{attribute 'GeneratedUsingTerminal: EL3773-0000-0019'}
{attribute addProperty BoxType "EL3773-0000-0019"}
{attribute addProperty Id "U1_SamplesAT %I*U1_Samples_2549228720"}
{attribute addProperty CRC "1101969407"}
{attribute addProperty Size "20"}
TYPE L1_Voltage_Samples_41AEB7FF :
STRUCT
	{attribute addProperty Name "U1_Samples"}
	U1_Samples AT %I* : U1_Samples_25492287;
END_STRUCT
END_TYPE

(* stored: Version 1.2.0.0, ProductVersion 3.1.4024.9
   DUT L1_Voltage_Samples_41AEB7FF: Id {1b4db75a-8035-4dfa-ab44-4667e4b49d13} *)
